// TwinCAT 3 PLC project Main
// ProgramVersion: 3.1.4024.0
// libraries:
//   Tc2_Standard, * (Beckhoff Automation GmbH)
//   Tc2_System, * (Beckhoff Automation GmbH)
//   Tc2_Utilities, * (Beckhoff Automation GmbH)
//   Tc3_Module, * (Beckhoff Automation GmbH)
//   TcUnit, * (www.tcunit.org)
//   mobject-graph,0.12.0,mobject
// project tree:
//   / PlcTask.TcTTO
//   POUs/ MAIN.TcPOU
//   Tests/Mocks/ TestNode.TcPOU (not stored)
//   Tests/ NodePrototype_TestSuite.TcPOU (not stored), NodeHost_TestSuite.TcPOU
// real-time tasks:
//   TASK PlcTask: cycle T#10ms, priority 20, ADS port 350

CONFIGURATION Main
    RESOURCE PLC ON TwinCAT3
        TASK PlcTask(INTERVAL := T#10ms, PRIORITY := 20);
        PROGRAM MAIN WITH PlcTask : MAIN;
    END_RESOURCE
END_CONFIGURATION

// ---- POUs/MAIN.TcPOU
PROGRAM MAIN
VAR
    nodeHost_TestSuite : NodeHost_TestSuite;
    nodePrototype_TestSuite : NodePrototype_TestSuite;
END_VAR

TcUnit.RUN();

END_PROGRAM

// ---- Tests/NodeHost_TestSuite.TcPOU
FUNCTION_BLOCK NodeHost_TestSuite EXTENDS TcUnit.FB_TestSuite
VAR
END_VAR

TestHasNodesAfterInit();
TestHasNodesAfterAdding();
TestRemoveNode();

METHOD TestHasNodesAfterAdding
VAR
    node : TestNode;
	host : NodeHost(0, 0);
	actual : BOOL;
END_VAR
TEST('TestHasNodesAfterAdding');

host.AddNode(Node);

actual := host.HasNodes;

AssertTrue(
	Condition := actual, 
	Message := 'Did not produce the expected result'
);

TEST_FINISHED();
END_METHOD

METHOD TestHasNodesAfterInit
VAR
	host : NodeHost(0, 0);
	actual : BOOL;
END_VAR
TEST('TestHasNodesAfterInit');

actual := host.HasNodes;

AssertFalse(
	Condition := actual, 
	Message := 'Did not produce the expected result'
);

TEST_FINISHED();
END_METHOD

METHOD TestRemoveNode
VAR CONSTANT
    NODES_TO_TEST : INT := 10;
END_VAR
VAR
    nodes : ARRAY [1..NODES_TO_TEST] OF TestNode;
    index : INT;
	host : NodeHost(0, 0);
	actual : BOOL;
END_VAR
TEST('TestRemoveNode');

FOR index := 1 TO NODES_TO_TEST BY 1 DO
    nodes[index].SetId(TO_STRING(index));
    host.AddNode(nodes[index]);
END_FOR

FOR index := 1 TO NODES_TO_TEST BY 1 DO
    host.RemoveNode(nodes[index]);
END_FOR

actual := host.HasNodes;

AssertFalse(
	Condition := actual, 
	Message := 'Did not produce the expected result'
);

TEST_FINISHED();
END_METHOD

END_FUNCTION_BLOCK
